% RSLogix 500 project Counter.RSS, saved by version 11.00.00.00 %
PROJECT "PHORP"    % processor: MicroLogix 1000 %

PROGRAM FILES
  LAD 2 "MAIN_PROG"  12 rungs
  LAD 3 "USER_FAULT"  1 rungs
  LAD 4 "HSC_INT"  1 rungs
  LAD 5 "STI_INT"  1 rungs
  LAD 6, 7, 8, 9, 10, 11, 12, 13, 14, 15, 16: only END

DATA FILES
  O0 OUTPUT  1 elements
  I1 INPUT  2 elements
  S2 STATUS  33 elements
  B3 BINARY  32 elements
  T4 TIMER  40 elements
  C5 COUNTER  32 elements
  R6 CONTROL  16 elements
  N7 INTEGER  105 elements

LADDER 2 "MAIN_PROG"
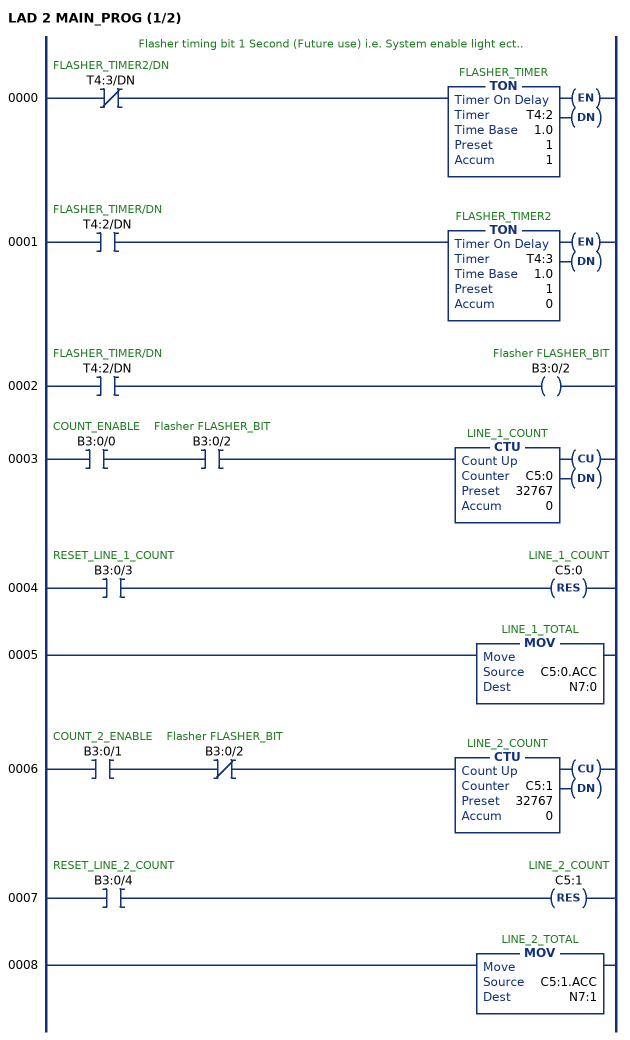
% Rung: 0 %
% Flasher timing bit 1 Second (Future use) i.e. System enable light ect.. %
SOR XIO T4:3/DN TON T4:2 1.0 1 1 EOR
%   T4:3  FLASHER_TIMER2 %
%   T4:2  FLASHER_TIMER %
% Rung: 1 %
SOR XIC T4:2/DN TON T4:3 1.0 1 0 EOR
%   T4:2  FLASHER_TIMER %
%   T4:3  FLASHER_TIMER2 %
% Rung: 2 %
SOR XIC T4:2/DN OTE B3:0/2 EOR
%   T4:2  FLASHER_TIMER %
%   B3:0/2  FLASHER_BIT  "Flasher" %
% Rung: 3 %
SOR XIC B3:0/0 XIC B3:0/2 CTU C5:0 32767 0 EOR
%   B3:0/0  COUNT_ENABLE %
%   B3:0/2  FLASHER_BIT  "Flasher" %
%   C5:0  LINE_1_COUNT %
% Rung: 4 %
SOR XIC B3:0/3 RES C5:0 EOR
%   B3:0/3  RESET_LINE_1_COUNT %
%   C5:0  LINE_1_COUNT %
% Rung: 5 %
SOR MOV C5:0.ACC N7:0 EOR
%   C5:0  LINE_1_COUNT %
%   N7:0  LINE_1_TOTAL %
% Rung: 6 %
SOR XIC B3:0/1 XIO B3:0/2 CTU C5:1 32767 0 EOR
%   B3:0/1  COUNT_2_ENABLE %
%   B3:0/2  FLASHER_BIT  "Flasher" %
%   C5:1  LINE_2_COUNT %
% Rung: 7 %
SOR XIC B3:0/4 RES C5:1 EOR
%   B3:0/4  RESET_LINE_2_COUNT %
%   C5:1  LINE_2_COUNT %
% Rung: 8 %
SOR MOV C5:1.ACC N7:1 EOR
%   C5:1  LINE_2_COUNT %
%   N7:1  LINE_2_TOTAL %

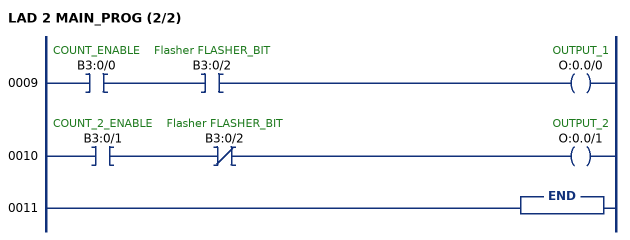
% Rung: 9 %
SOR XIC B3:0/0 XIC B3:0/2 OTE O:0.0/0 EOR
%   B3:0/0  COUNT_ENABLE %
%   B3:0/2  FLASHER_BIT  "Flasher" %
%   O:0.0/0  OUTPUT_1 %
% Rung: 10 %
SOR XIC B3:0/1 XIO B3:0/2 OTE O:0.0/1 EOR
%   B3:0/1  COUNT_2_ENABLE %
%   B3:0/2  FLASHER_BIT  "Flasher" %
%   O:0.0/1  OUTPUT_2 %
% Rung: 11 %
SOR END EOR

OTHER DOCUMENTED ADDRESSES
  I:0.0/0  SYSTEM_ENABLE

DATA TABLE (non-zero values as saved)
DATA T4
% .PRE .ACC %
% T4:1 % 50 0
% T4:2 % 1 1
% T4:3 % 1 0
% T4:4 % 100 0
% T4:5 % 100 0
% T4:6 % 200 0
DATA C5
% .PRE .ACC %
% C5:0 % 32767 0
% C5:1 % 32767 0
